Fanuc KAREL source: kd00047.KL

-- PROVISIONAL review KL for V770-1; original PC SHA256 ef29852811a8bbd47e05f5a03cb31d4414c0472509dad3ae7502e1b6ce67e2dd
-- Incomplete behavior may be omitted. Consult companion uncertainty JSON. Do not deploy.
PROGRAM KD00047
%NOLOCKGROUP
VAR
  I : INTEGER
  J : INTEGER
  B : BOOLEAN
  R : REAL
  S : STRING[80]
-- UNRESOLVED_DECL V type=000013
BEGIN
  -- UNRESOLVED_PC offsets 5-20; opcodes 2E,22,32,35
  -- UNRESOLVED_PC offsets 25-46; opcodes 01,49,2E,0A,82,0B
  -- UNRESOLVED_PC offsets 51-55; opcodes 7F
END KD00047
